{attribute 'GeneratedUsingTerminal: EP3182-1002-0018'}
{attribute addProperty BoxType "EP3182-1002-0018"}
{attribute addProperty Id "EtcSlaveTerminalBaseAI_Standard_Channel_1AT %I*AI_Standard_Channel_A8DF64E310AI_Standard_Channel_2AT %I*AI_Standard_Channel_A8DF64E310DO_OutputsAT %Q*DO_Outputs_C0F4C3832WcStateAT %I*WcState_9091E0EB2InfoDataAT %I*InfoData_32EB74EA10"}
{attribute addProperty CRC "1002784816"}
{attribute addProperty Size "34"}
TYPE EP3182_3BC54830 EXTENDS EtcSlaveTerminalBase :
STRUCT
	{attribute addProperty Name "AI_Standard_Channel_1"}
	AI_Standard_Channel_1 : AI_Standard_Channel_A8DF64E3;
	{attribute addProperty Name "AI_Standard_Channel_2"}
	AI_Standard_Channel_2 : AI_Standard_Channel_A8DF64E3;
	{attribute addProperty Name "DO_Outputs"}
	DO_Outputs : DO_Outputs_C0F4C383;
	{attribute addProperty Name "WcState"}
	WcState : WcState_9091E0EB;
	{attribute addProperty Name "InfoData"}
	InfoData : InfoData_32EB74EA;
END_STRUCT
END_TYPE

(* stored: Version 1.2.0.0, ProductVersion 3.1.4024.9
   DUT EP3182_3BC54830: Id {cd78e795-d950-40a9-b52d-f3d749d3bd89} *)
